{attribute 'Tc2GvlVarNames'}
VAR_GLOBAL CONSTANT
	(* KKWW_Zustand_Status *)
	E_MVWW_Zustand_Status_Idle_Sperre				: SINT := 0;
	E_MVWW_Zustand_Status_Betriebsbereit			: SINT := 1;
	E_MVWW_Zustand_Status_Nachl					: SINT := 2;
	E_MVWW_Zustand_Status_Vorl						: SINT := 3;
	E_MVWW_Zustand_Status_Betrieb					: SINT := 4;
	E_MVWW_Zustand_Status_Betrieb_Sperre			: SINT := 5;
	E_MVWW_Zustand_Status_Stoerung				: SINT := 99;

	(* System_KKWW_Zustand_Status *)
	E_System_MVWW_Zustand_Status_Idle_Sperre		: SINT := 0;
	E_System_MVWW_Zustand_Status_Betriebsbereit		: SINT := 1;
	E_System_MVWW_Zustand_Status_Nachl_Stellventil	: SINT := 2;
	E_System_MVWW_Zustand_Status_Vorl_Stellventil	: SINT := 3;
	E_System_MVWW_Zustand_Status_Nachl_Pumpe		: SINT := 4;
	E_System_MVWW_Zustand_Status_Vorl_Pumpe		: SINT := 5;
	(*E_System_MVWW_Zustand_Status_Nachl_KKWW		: SINT := 6;
	E_System_MVWW_Zustand_Status_Vorl_KKWW			: SINT := 7;	*)
	E_System_MVWW_Zustand_Status_Betrieb			: SINT := 8;
	E_System_MVWW_Zustand_Status_Betrieb_Sperre	: SINT := 9;
	E_System_MVWW_Zustand_Status_Stoerung			: SINT := 99;
END_VAR

(* stored: Version 1.1.0.1, ProductVersion 3.1.4024.9
   GVL Con_MVWW: Id {f148344a-d9c2-4393-b5fa-7097b2c7af36} *)
